{region '#Template'}
	{attribute 'Version' := '5.1.0.0'}
	{attribute 'Tags' := '"LCID": "1031", "Text": "Gebäudeautomation, Einbruchalarm"'}
	{attribute 'Tags' := '"LCID": "1033", "Text": "Building automation, Burglar alarm"'}
	{attribute 'Using' := '"Type": "Template", "URI": "BA2_Param"'}
	{attribute 'Using' := '"Type": "Template", "URI": "Site"'}		 
	{attribute 'Using' := '"Type": "Template", "URI": "EC_ID"'}
	{attribute 'Using' := '"Type": "Template", "URI": "ST_BA_BuildingAlarms"'}
	{attribute 'Description' := '"LCID": "1031", "Text": "Gebäude Einbruchalarm"'}
	{attribute 'Description' := '"LCID": "1033", "Text": "Building Burglar alarm"'}
{endregion}
FUNCTION_BLOCK FB_BA_BurglarAlarmSystem EXTENDS FB_BA_View
VAR_INPUT CONSTANT
	MagneticContact01		: FB_BA_SensorBinary;                      
END_VAR

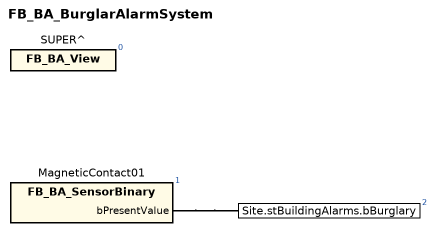
SUPER^(); // FB_BA_View
MagneticContact01(); // FB_BA_SensorBinary
Site.stBuildingAlarms.bBurglary := MagneticContact01.bPresentValue;

METHOD FB_init : BOOL
VAR_INPUT
	bInitRetains	: BOOL; // if TRUE, the retain variables are initialized (warm start / cold start)
	bInCopyCode		: BOOL;  // if TRUE, the instance afterwards gets moved into the copy code (online change)
END_VAR
MagneticContact01.iParent				:= THIS^;	
MagneticContact01.iLabel				:= LblCtl_MagneticSwitch;
MagneticContact01.eDPADMode				:= E_BA_DPADMode.eInclude;
MagneticContact01.Input.iLabel			:= LblFun_DangerAlarm;
MagneticContact01.Input.sObjectName		:= '{Idx=41}';
MagneticContact01.Input.nEventClassID	:= EC_ID.NC10;
MagneticContact01.Input.ePolarity		:= E_BA_Polarity.eReverse;
MagneticContact01.Input.eEnPlantLock	:= E_BA_LockPriority.eNoLock;
END_METHOD

END_FUNCTION_BLOCK

(* stored: Version 1.1.0.1, ProductVersion 3.1.4024.12
   POU FB_BA_BurglarAlarmSystem: Id {428c168c-235c-4f6a-8ab5-e4a3fc37871a}, SpecialFunc None
   Method FB_init: Id {d947fbbf-f259-4234-b03b-cd08464c02fb} *)
